TYPE ST_OutfeedConfig :
	STRUCT
	END_STRUCT
END_TYPE

(* stored: Version 1.1.0.1, ProductVersion 3.1.4024.12
   DUT ST_OutfeedConfig: Id {a1ee704e-b6d0-4e50-8d9c-c5e1a8d30a51} *)
